# EPICS autosave request: utcaApp/Db/trigger_iface_channel.req
$(P)$(R)$(TRIGGER_NAME)$(TRIGGER_CHAN)Dir-Sel
$(P)$(R)$(TRIGGER_NAME)$(TRIGGER_CHAN)DirPol-Sel
$(P)$(R)$(TRIGGER_NAME)$(TRIGGER_CHAN)RcvLen-SP
$(P)$(R)$(TRIGGER_NAME)$(TRIGGER_CHAN)TrnLen-SP
